RoboDK station: RobotStationFlatSurface.rdk

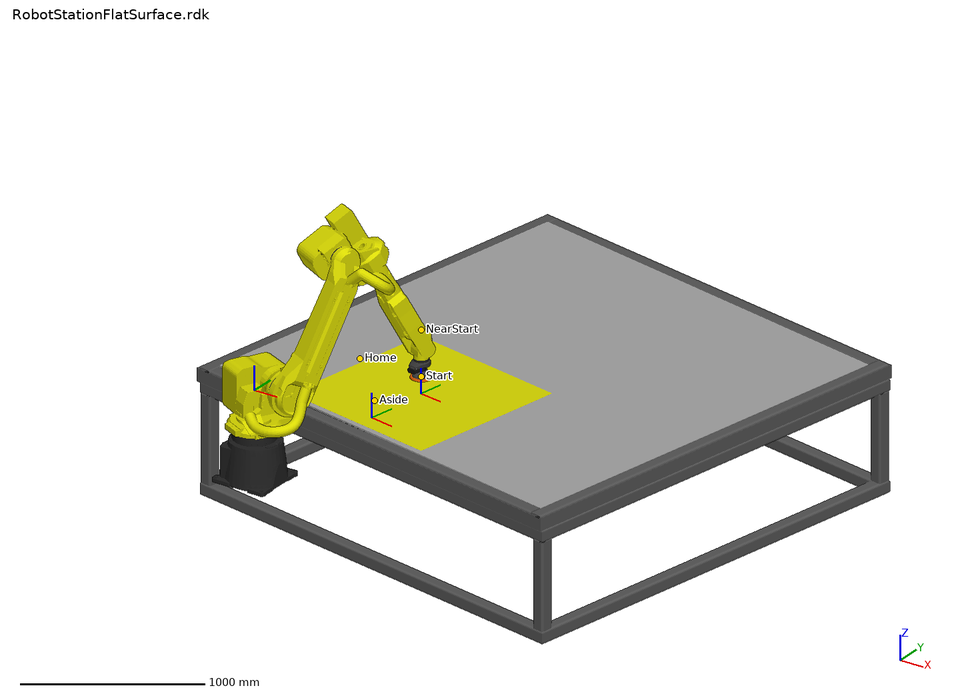
[picture v0: the station drawn from its stored meshes, robots at their saved joint values, targets as dots, program paths as lines]
Station RobotStationFlatSurface (saved by RoboDK 5.1.1). Poses are relative to the parent item; angles as X-Y-Z fixed-axis rotations.
  - frame Fanuc M-20iA/35M Base at (-96.84, 0, 525) mm
    - robot Fanuc M-20iA/35M: 6 axes, payload 35 kg, reach 1813 mm, repeatability 0.04 mm, weight 252 kg
        modified DH rows (alpha deg, a mm, theta deg, d mm): 0, 0, 0, 525; -90, 150, -90, 0; 0, 790, 0, 0; -90, 150, 0, 860; 90, 0, 0, 0; -90, 0, 0, 100
        base shift (0, 0, -525) mm
        joint limits [-185, -110, -85, -200, -190, -450] to [185, 110, 245, 200, 190, 450]; home [0, 0, 0, 0, 0, 0]; saved at [64.344, 25.651, -61.694, 180, 28.306, -254.344]
      - tool RobotiQ Sanding Kit, TCP at (0, 0, 90.86) mm, size 127 x 139.7 x 103.3 mm
  - frame ObjectFrame at (349.91, 930.11, 260.24) mm, rotated rx 0 ry 0 rz -10 deg
    - object Plane 1m x 1m at (0, 0, 0) mm, size 1000 x 1000 x 0.5 mm, geometry from plane_1m.sld
    - target Aside (Cartesian target) at (431.99, -785.44, 374.27) mm, rotated rx -90 ry 0 rz -90 deg; joints [11.829, -11.383, -59.508, -24.931, 61.898, -77.649] of Fanuc M-20iA/35M
    - target Home (Cartesian target) at (14.25, -478.75, 379.42) mm, rotated rx -90 ry 0 rz 0 deg; joints [37.9, -26.83, -52.44, -131.261, -63.108, 62.726] of Fanuc M-20iA/35M
    - target NearStart (Cartesian target) at (1.18, 1.36, 379) mm, rotated rx -180 ry 0 rz 0 deg; joints [64.301, 10.823, -42.533, 180, 47.467, -254.301] of Fanuc M-20iA/35M
    - target Start (Cartesian target) at (0, 0, 100) mm, rotated rx -180 ry 0 rz 0 deg; joints [64.344, 25.651, -61.694, -180, 28.306, 105.656] of Fanuc M-20iA/35M
  - frame TableFrame at (-612.8, 1841.55, -520.07) mm, rotated rx 0 ry 0 rz -10.03 deg
    - object Table 108x114x32 IN at (0, 0, 0) mm, size 2628.9 x 2679.7 x 778.4 mm, geometry from Table-108x114x32-IN.sld
